FUNCTION_BLOCK DataPanel_MI_QXA (* Composite FB for boolean output data *)
  (* Standard: 61499-2; Description: Copyright (c) 2024 HR Agrartechnik GmbH This program and the accompanying materials are made available under the terms of the Eclipse Public License 2.0 which is available at https://www.eclipse.org/legal/epl-2.0/ SPDX-License-Identifier: EPL-2.0 *)
  (* Version 1.0, 2024-04-24, Franz Höpfinger, HR Agrartechnik GmbH *)
  PACKAGE DataPanel::io::MI::DQ;
  IMPORT DataPanel::io::MI::DQ::DataPanel_MI_DO::Invalid;
  IMPORT DataPanel::io::MI::const::MI;
  IMPORT eclipse4diac::core::TypeHash;
  (* Documentation:
  Copyright (c) 2024 HR Agrartechnik GmbH   
   This program and the accompanying materials are made    
   available under the terms of the Eclipse Public License 2.0    
   which is available at https://www.eclipse.org/legal/epl-2.0/    
   SPDX-License-Identifier: EPL-2.0
  *)
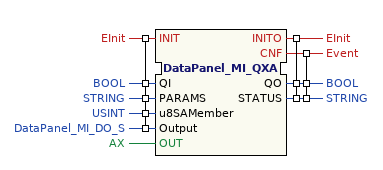
  EVENT_INPUT
    INIT : EInit WITH QI, PARAMS, u8SAMember, Output; (* Service Initialization *)
  END_EVENT
  EVENT_OUTPUT
    INITO : EInit WITH QO, STATUS; (* Initialization Confirm *)
    CNF WITH QO, STATUS; (* Confirmation of Requested Service *)
  END_EVENT
  VAR_INPUT
    QI : BOOL; (* Event Input Qualifier *)
    PARAMS : STRING; (* Service Parameters *)
    u8SAMember : USINT := MI::MI_00; (* Node SA 224..239 *)
    Output : DataPanel::io::MI::DQ::DataPanel_MI_DO_S := Invalid; (* Identify the Output DigitalOutput_1A..8B and Input_Power_Port_5..8 *)
  END_VAR
  VAR_OUTPUT
    QO : BOOL; (* Event Output Qualifier *)
    STATUS : STRING; (* Service Status *)
  END_VAR
  SOCKETS
    OUT : adapter::types::unidirectional::AX;
  END_SOCKETS
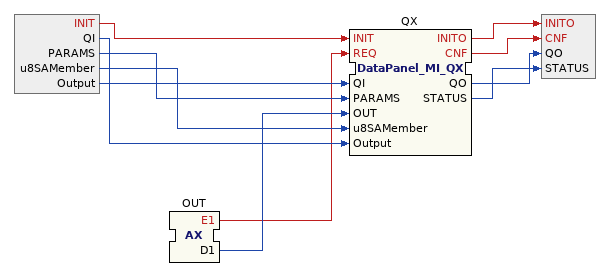
  FBS
    QX : DataPanel::io::MI::DQ::DataPanel_MI_QX;
  END_FBS
  EVENT_CONNECTIONS
    INIT TO QX.INIT;
    QX.INITO TO INITO;
    OUT.E1 TO QX.REQ;
    QX.CNF TO CNF;
  END_CONNECTIONS
  DATA_CONNECTIONS
    OUT.D1 TO QX.OUT;
    QI TO QX.QI;
    PARAMS TO QX.PARAMS;
    QX.QO TO QO;
    QX.STATUS TO STATUS;
    u8SAMember TO QX.u8SAMember;
    Output TO QX.Output;
  END_CONNECTIONS
END_FUNCTION_BLOCK
